PROGRAM Operation
VAR
	TON_0: TON;
	TON_1: TON;
	StopMemory :BOOL;
END_VAR
VAR // added by the converter: edge detectors and wires of the graphical bodies
    _w1 : BOOL;
END_VAR

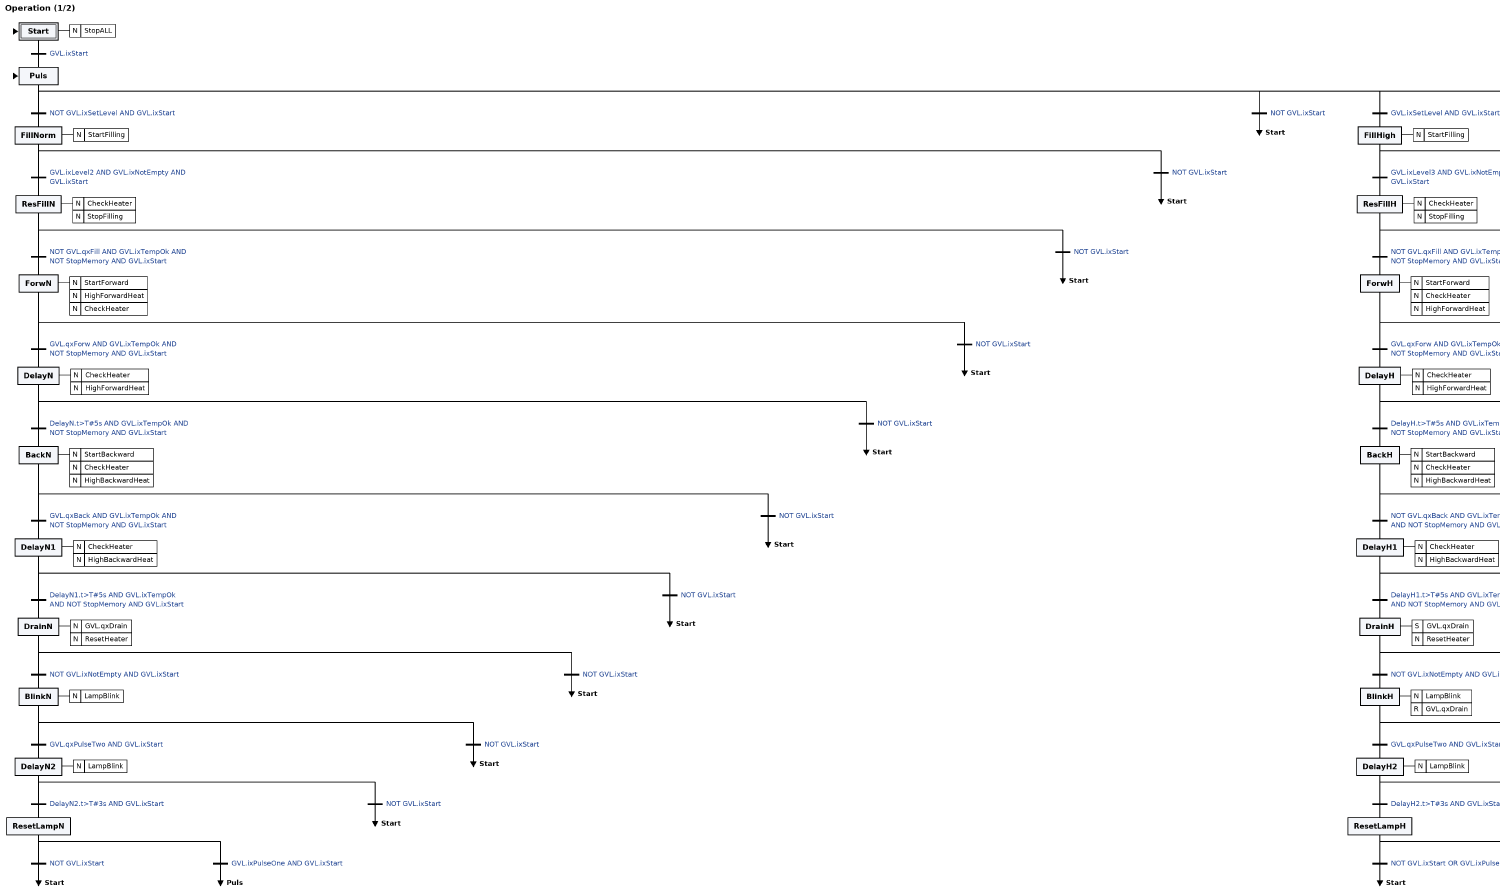
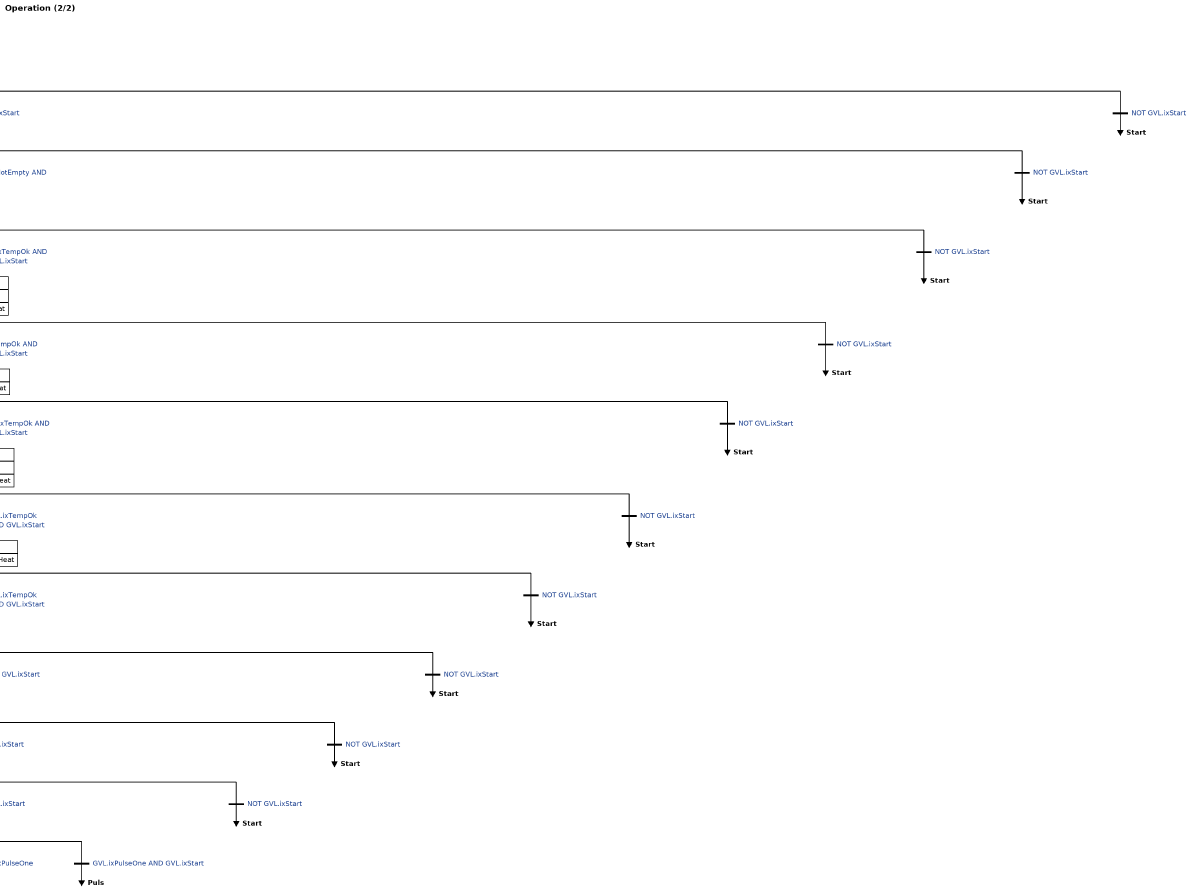
INITIAL_STEP Start:
    StopALL(N);
END_STEP
TRANSITION FROM Start TO Puls
    := GVL.ixStart;
END_TRANSITION
STEP Puls:
END_STEP
TRANSITION FROM Puls TO FillNorm
    := NOT GVL.ixSetLevel AND GVL.ixStart;
END_TRANSITION
TRANSITION FROM Puls TO Start
    := NOT GVL.ixStart;
END_TRANSITION
STEP FillNorm:
    StartFilling(N);
END_STEP
TRANSITION FROM FillNorm TO ResFillN
    := GVL.ixLevel2 AND GVL.ixNotEmpty AND GVL.ixStart;
END_TRANSITION
TRANSITION FROM FillNorm TO Start
    := NOT GVL.ixStart;
END_TRANSITION
STEP ResFillN:
    CheckHeater(N);
    StopFilling(N);
END_STEP
TRANSITION FROM ResFillN TO ForwN
    := NOT GVL.qxFill AND GVL.ixTempOk AND NOT StopMemory AND GVL.ixStart;
END_TRANSITION
TRANSITION FROM ResFillN TO Start
    := NOT GVL.ixStart;
END_TRANSITION
STEP ForwN:
    StartForward(N);
    HighForwardHeat(N);
    CheckHeater(N);
END_STEP
TRANSITION FROM ForwN TO DelayN
    := GVL.qxForw AND GVL.ixTempOk AND NOT StopMemory AND GVL.ixStart;
END_TRANSITION
TRANSITION FROM ForwN TO Start
    := NOT GVL.ixStart;
END_TRANSITION
STEP DelayN:
    CheckHeater(N);
    HighForwardHeat(N);
END_STEP
TRANSITION FROM DelayN TO BackN
    := DelayN.t>T#5s AND GVL.ixTempOk AND NOT StopMemory AND GVL.ixStart;
END_TRANSITION
TRANSITION FROM DelayN TO Start
    := NOT GVL.ixStart;
END_TRANSITION
STEP BackN:
    StartBackward(N);
    CheckHeater(N);
    HighBackwardHeat(N);
END_STEP
TRANSITION FROM BackN TO DelayN1
    := GVL.qxBack AND GVL.ixTempOk AND NOT StopMemory AND GVL.ixStart;
END_TRANSITION
TRANSITION FROM BackN TO Start
    := NOT GVL.ixStart;
END_TRANSITION
STEP DelayN1:
    CheckHeater(N);
    HighBackwardHeat(N);
END_STEP
TRANSITION FROM DelayN1 TO DrainN
    := DelayN1.t>T#5s AND GVL.ixTempOk AND NOT StopMemory AND GVL.ixStart;
END_TRANSITION
TRANSITION FROM DelayN1 TO Start
    := NOT GVL.ixStart;
END_TRANSITION
STEP DrainN:
    GVL.qxDrain(N);
    ResetHeater(N);
END_STEP
TRANSITION FROM DrainN TO BlinkN
    := NOT GVL.ixNotEmpty AND GVL.ixStart;
END_TRANSITION
TRANSITION FROM DrainN TO Start
    := NOT GVL.ixStart;
END_TRANSITION
STEP BlinkN:
    LampBlink(N);
END_STEP
TRANSITION FROM BlinkN TO DelayN2
    := GVL.qxPulseTwo AND GVL.ixStart;
END_TRANSITION
TRANSITION FROM BlinkN TO Start
    := NOT GVL.ixStart;
END_TRANSITION
STEP DelayN2:
    LampBlink(N);
END_STEP
TRANSITION FROM DelayN2 TO ResetLampN
    := DelayN2.t>T#3s AND GVL.ixStart;
END_TRANSITION
TRANSITION FROM DelayN2 TO Start
    := NOT GVL.ixStart;
END_TRANSITION
STEP ResetLampN:
END_STEP
TRANSITION FROM ResetLampN TO Start
    := NOT GVL.ixStart;
END_TRANSITION
TRANSITION FROM ResetLampN TO Puls
    := GVL.ixPulseOne AND GVL.ixStart;
END_TRANSITION
TRANSITION FROM Puls TO FillHigh
    := GVL.ixSetLevel AND GVL.ixStart;
END_TRANSITION
TRANSITION FROM Puls TO Start
    := NOT GVL.ixStart;
END_TRANSITION
STEP FillHigh:
    StartFilling(N);
END_STEP
TRANSITION FROM FillHigh TO ResFillH
    := GVL.ixLevel3 AND GVL.ixNotEmpty AND GVL.ixStart;
END_TRANSITION
TRANSITION FROM FillHigh TO Start
    := NOT GVL.ixStart;
END_TRANSITION
STEP ResFillH:
    CheckHeater(N);
    StopFilling(N);
END_STEP
TRANSITION FROM ResFillH TO ForwH
    := NOT GVL.qxFill AND GVL.ixTempOk AND NOT StopMemory AND GVL.ixStart;
END_TRANSITION
TRANSITION FROM ResFillH TO Start
    := NOT GVL.ixStart;
END_TRANSITION
STEP ForwH:
    StartForward(N);
    CheckHeater(N);
    HighForwardHeat(N);
END_STEP
TRANSITION FROM ForwH TO DelayH
    := GVL.qxForw AND GVL.ixTempOk AND NOT StopMemory AND GVL.ixStart;
END_TRANSITION
TRANSITION FROM ForwH TO Start
    := NOT GVL.ixStart;
END_TRANSITION
STEP DelayH:
    CheckHeater(N);
    HighForwardHeat(N);
END_STEP
TRANSITION FROM DelayH TO BackH
    := DelayH.t>T#5s AND GVL.ixTempOk AND NOT StopMemory AND GVL.ixStart;
END_TRANSITION
TRANSITION FROM DelayH TO Start
    := NOT GVL.ixStart;
END_TRANSITION
STEP BackH:
    StartBackward(N);
    CheckHeater(N);
    HighBackwardHeat(N);
END_STEP
TRANSITION FROM BackH TO DelayH1
    := NOT GVL.qxBack AND GVL.ixTempOk AND NOT StopMemory AND GVL.ixStart;
END_TRANSITION
TRANSITION FROM BackH TO Start
    := NOT GVL.ixStart;
END_TRANSITION
STEP DelayH1:
    CheckHeater(N);
    HighBackwardHeat(N);
END_STEP
TRANSITION FROM DelayH1 TO DrainH
    := DelayH1.t>T#5s AND GVL.ixTempOk AND NOT StopMemory AND GVL.ixStart;
END_TRANSITION
TRANSITION FROM DelayH1 TO Start
    := NOT GVL.ixStart;
END_TRANSITION
STEP DrainH:
    GVL.qxDrain(S);
    ResetHeater(N);
END_STEP
TRANSITION FROM DrainH TO BlinkH
    := NOT GVL.ixNotEmpty AND GVL.ixStart;
END_TRANSITION
TRANSITION FROM DrainH TO Start
    := NOT GVL.ixStart;
END_TRANSITION
STEP BlinkH:
    LampBlink(N);
    GVL.qxDrain(R);
END_STEP
TRANSITION FROM BlinkH TO DelayH2
    := GVL.qxPulseTwo AND GVL.ixStart;
END_TRANSITION
TRANSITION FROM BlinkH TO Start
    := NOT GVL.ixStart;
END_TRANSITION
STEP DelayH2:
    LampBlink(N);
END_STEP
TRANSITION FROM DelayH2 TO ResetLampH
    := DelayH2.t>T#3s AND GVL.ixStart;
END_TRANSITION
TRANSITION FROM DelayH2 TO Start
    := NOT GVL.ixStart;
END_TRANSITION
STEP ResetLampH:
END_STEP
TRANSITION FROM ResetLampH TO Start
    := NOT GVL.ixStart OR GVL.ixPulseOne;
END_TRANSITION
TRANSITION FROM ResetLampH TO Puls
    := GVL.ixPulseOne AND GVL.ixStart;
END_TRANSITION

ACTION CheckHeater:
IF GVL.iwCurrentTemp < GVL.iwSetTemp AND NOT StopMemory THEN
	GVL.qxHeatingON :=TRUE;
	
ELSIF StopMemory AND GVL.iwCurrentTemp > GVL.iwSetTemp THEN
	GVL.qxHeatingON := FALSE;
END_IF

IF GVL.iwCurrentTemp +4 > GVL.iwSetTemp THEN
	StopMemory := TRUE;
ELSE
	StopMemory := FALSE;
END_IF


IF (GVL.iwCurrentTemp = GVL.iwSetTemp - 3) OR (GVL.iwCurrentTemp = GVL.iwSetTemp - 2) OR (GVL.iwCurrentTemp = GVL.iwSetTemp - 1) OR (GVL.iwCurrentTemp = GVL.iwSetTemp) THEN
	GVL.ixTempOk := TRUE;
	StopMemory := FALSE;
END_IF

IF (GVL.iwCurrentTemp = GVL.iwSetTemp + 3) OR (GVL.iwCurrentTemp = GVL.iwSetTemp + 2) OR (GVL.iwCurrentTemp = GVL.iwSetTemp + 1) OR (GVL.iwCurrentTemp = GVL.iwSetTemp) THEN
	GVL.ixTempOk := TRUE;
	StopMemory := FALSE;
END_IF
END_ACTION

ACTION DrainStopHeat:
IF StopMemory=TRUE THEN
	GVL.qxDrain:=FALSE;
ELSE
	GVL.qxForw:=TRUE;
END_IF
END_ACTION

ACTION HighBackwardHeat:
IF StopMemory=TRUE THEN
	GVL.qxBack:=FALSE;
ELSE
	GVL.qxBack:=TRUE;
END_IF
END_ACTION

ACTION HighForwardHeat:
IF StopMemory=TRUE THEN
	GVL.qxForw:=FALSE;
ELSE
	GVL.qxForw:=TRUE;
END_IF
END_ACTION

ACTION LampBlink:
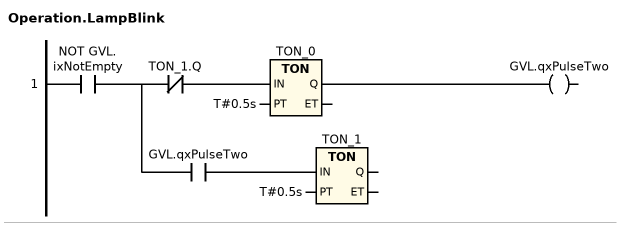
// NETWORK 1
_w1 := NOT GVL.ixNotEmpty;
TON_0(IN := _w1 AND NOT TON_1.Q, PT := T#0.5s); // TON
GVL.qxPulseTwo := TON_0.Q;
TON_1(IN := _w1 AND GVL.qxPulseTwo, PT := T#0.5s); // TON
END_ACTION

ACTION ResetHeater:
GVL.qxHeatingON := FALSE;
GVL.qxBack := FALSE;
END_ACTION

ACTION StartBackward:
GVL.qxBack := TRUE;
GVL.qxForw := FALSE;
END_ACTION

ACTION StartFilling:
GVL.qxFill := TRUE;
GVL.qxDrain := FALSE;
END_ACTION

ACTION StartForward:
GVL.qxForw := TRUE;
GVL.qxBack := FALSE;
END_ACTION

ACTION StopALL:
GVL.qxFill := FALSE;
GVL.qxForw := FALSE;
GVL.qxBack := FALSE;
GVL.qxDrain := TRUE;
GVL.qxHeatingON := FALSE;
END_ACTION

ACTION StopFilling:
GVL.qxFill := FALSE;
END_ACTION

END_PROGRAM

(* stored: Version 1.1.0.1, ProductVersion 3.1.4024.12
   POU Operation: Id {43472cc5-ea16-4feb-adef-51b77ade00d6}, SpecialFunc None
   Action CheckHeater: Id {79a1ac9a-4a34-4a20-b1ff-5a6c675999cd}
   Action DrainStopHeat: Id {452ffdc5-5930-4049-b073-7ac7a4b24dce}
   Action HighBackwardHeat: Id {ecc2944a-de39-4d54-9286-f609255e150c}
   Action HighForwardHeat: Id {f65243b3-17eb-48b3-b66b-d520041cb405}
   Action LampBlink: Id {b8e3407f-79ee-4510-8ddc-6dfd27031bb6}
   Action ResetHeater: Id {18843537-5f7e-4110-855a-72f409682fe3}
   Action StartBackward: Id {86ba261f-6c3a-461b-a86f-df2363ef3124}
   Action StartFilling: Id {56ff99fd-c365-453e-87bc-dacc30b538f0}
   Action StartForward: Id {7fc9b6d3-011e-4092-8bc8-7e2ddadaf64d}
   Action StopALL: Id {e57881e4-c433-4614-a7de-2fbb50efa70a}
   Action StopFilling: Id {2fad9aa2-5167-4ac4-ab20-623a8b406346} *)
